TYPE EL3443_TotalBasic :
STRUCT
	{attribute addProperty Name "Frequency"}
	Frequency AT %I* : REAL;
	{attribute addProperty Name "Power Factor"}
	PowerFactor AT %I* : REAL;
	{attribute addProperty Name "Calculated Neutral Line Current"}
	CalculatedNeutralLineCurrent AT %I* : REAL;
END_STRUCT
END_TYPE

(* stored: Version 1.1.0.1, ProductVersion 3.1.4024.9
   DUT EL3443_TotalBasic: Id {f74b33b5-2ee3-0ddc-1e9b-1f7df2958c12} *)
